(* PLC project v0.6.02_RefactorGateAndTest.project, CODESYS CODESYS V3.5 SP19 Patch 1 *)
(* stored: creationDateTime 2026-08-15T01:12:17.402982, modificationDateTime 2026-08-15T01:12:17.402982 *)

(* ═══════════════════════════════════════════════════════════════ ⚙️ ST_MotionChecklist — Diagnostic chronologique de commande de mouvement ─────────────────────────────────────────────────────────────── 🎨 Permet de voir en un coup d'œil pourquoi un ordre de mouvement ne fait pas coller les relais. ═══════════════════════════════════════════════════════════════ *)
TYPE ST_MotionChecklist : STRUCT
  Step1_PowerEngaged : BOOL;  (* 1. Puissance & Mode TRUE = Contacteur principal sous tension (PowerContactorEngaged_DI) ➔ Armer puissance via Reset *)
  Step2_ModeAuthorized : BOOL;  (* TRUE = Mode MAINT_N1 ou N2 actif (pas DISABLE) ➔ Commutateur Mode IHM *)
  Step3_NotBusyOtherTask : BOOL;  (* TRUE = Pas d'autre séquence en cours (Homing, Benne busy, etc.) *)
  HwIn_PowerContactorEngaged_DI : BOOL;  (* 1bis. Entrées physiques directes HwIn (vérité terrain) Contacteur puissance principal issu de HwIn.Machine *)
  HwIn_BrakeIsOpen_DI : BOOL;  (* Retour fin de course frein (1 = ouvert) issu de HwIn *)
  Cmd_BrakeRelease : BOOL;  (* Ordre de commande d'ouverture de frein généré par l'automate *)
  Step4_MotionRequested : BOOL;  (* 2. Intention & Demande TRUE = Demande active (Bouton IHM ou Joystick) ➔ Si IHM : TglJoystickMaster doit être à 0 ! *)
  RequestedDirection : INT;  (* +1 = Montée, -1 = Descente, 0 = Repos *)
  RequestedSpeedPct : REAL;  (* 0..100 % consigne demandée *)
  Step5_NoSafetyFault : BOOL;  (* 3. Chaîne de Sécurité & Verrous TRUE = Pas de SafeStop ni AU actif sur cet axe *)
  Step6_DirectionAllowed : BOOL;  (* TRUE = Sens autorisé (AscentPermit/DescendPermit) *)
  Step7_BrakeReleased : BOOL;  (* TRUE = Commande frein activée & retour frein OK *)
  Step8_OutputInterlockOk : BOOL;  (* TRUE = Étage de sortie LD débloqué (pas d'interlock actif) *)
  AllConditionsMet : BOOL;  (* 4. Bilan & Exécution Physiques 🟢 TRUE = TOUTES LES CONDITIONS SONT REMPLIES, LES RELAIS DOIVENT COLLER ! *)
  RelayFwdActive : BOOL;  (* 🛗 Relais Montée physiquement commandé *)
  RelayRevActive : BOOL;  (* 🛗 Relais Descente physiquement commandé *)
  SpeedContactor1Active : BOOL;  (* 🔌 Contacteur de vitesse Palier 1 commandé *)
END_STRUCT;
END_TYPE
